{attribute 'qualified_only'}
{attribute 'strict'}
{attribute 'to_string'}
//定义命令、运动状态
TYPE E_AxisCommand :
(
    NoCommand    := 0,    // 当前没有运动命令

    PowerOn      := 10,   // 请求轴使能
    PowerOff     := 20,   // 请求轴撤销使能
    Reset        := 30,   // 轴错误复位
    Stop         := 40,   // 软件停止
	Halt		 := 50,	  // 减速停止
    Home         := 60,   // 回零
	
    MoveRelative := 70,   // 相对运动
    MoveAbsolute := 80,   // 绝对运动
	JogPositive  := 90,	  // 正向点动
	JogNegative  := 100,  // 反向点动
	
	TorqueControl:= 110   // 力矩模式
);
END_TYPE

(* stored: Version 1.1.0.1, ProductVersion 3.1.4026.18
   DUT E_AxisCommand: Id {4e6d8c7c-13c7-415d-a8df-33d2cc40a365} *)
